(* PLC project CoDeSys External Library Template, WAGO e!COCKPIT e!COCKPIT, author 3S - Smart Software Solutions GmbH *)
(* stored: creationDateTime 2019-10-29T12:22:40.8522817, version 3.5.5.30, modificationDateTime 2019-10-24T14:40:07.960949, organization 3S - Smart Software Solutions GmbH *)
(* Library project template with all possible element types, docu and a sample project structure *)

FUNCTION fnKomunikatDaneErrorRetry : STRING
  VAR_INPUT
    xAktywny : BOOL;
    intKlasa : INT;
    intNumer : INT;
  END_VAR
  VAR
    sDane : alSTRINGKomunikat;
    typKomunikat : typKomunikat;
  END_VAR

            (* funkcja tylko dla reakcji na Q *)

IF xAktywny THEN
	sDane := CONCAT('RETRY=1;ACT=1;CLASS=' , INT_TO_STRING(intKlasa));
	ELSE
	sDane := CONCAT('RETRY=1;ACT=0;CLASS=' , INT_TO_STRING(intKlasa));	
END_IF
sDane := CONCAT(sDane , ';NUM=');	
sDane := CONCAT(sDane , INT_TO_STRING(intNumer));
sDane := CONCAT(sDane , ';E');
sDane := CONCAT(sDane , fnKonwersjaINT_STRING(intWartosc := intNumer , intIloscZnakow := 3));
IF xAktywny THEN
	sDane := CONCAT(sDane, 'ACT=1');
	ELSE
	sDane := CONCAT(sDane, 'ACT=0');
END_IF
fnKomunikatDaneErrorRetry := sDane;

          
END_FUNCTION
